FUNCTION_BLOCK ReservatorioElevado (* Composite Function Block Type *)
  (* Standard: 61499-2 *)
  (* Version 0.0, 02/03/2026, template *)
  PACKAGE Hidryco.HidrycoLib;
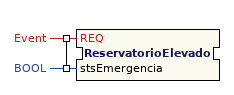
  EVENT_INPUT
    REQ WITH stsEmergencia;
  END_EVENT
  VAR_INPUT
    stsEmergencia : BOOL;
  END_VAR
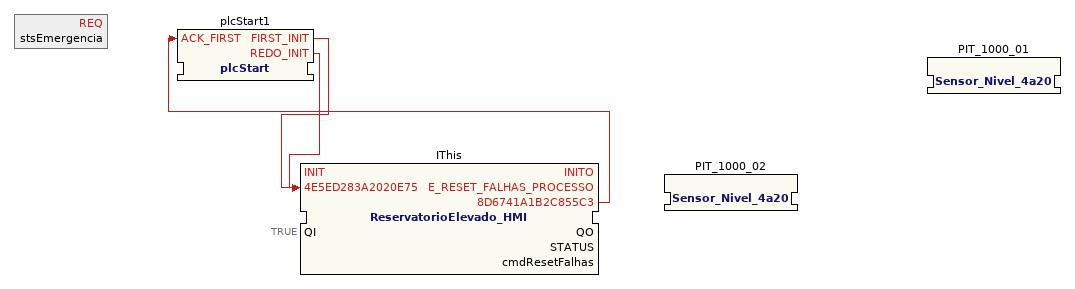
  FBS
    PIT_1000_02 : Sensor_Nivel_4a20;
    PIT_1000_01 : Sensor_Nivel_4a20;
    IThis : ReservatorioElevado_HMI(QI := TRUE);
    plcStart1 : plcStart;
  END_FBS
  EVENT_CONNECTIONS
    plcStart1.FIRST_INIT TO IThis.4E5ED283A2020E75;
    plcStart1.REDO_INIT TO IThis.4E5ED283A2020E75;
    IThis.8D6741A1B2C855C3 TO plcStart1.ACK_FIRST;
  END_CONNECTIONS
END_FUNCTION_BLOCK
